FUNCTION WORDS_TO_ARR08B_BE (* this Function combines 4 WORDSs to a 8-BYTE Array; Big-Endian-Format (Network Byte Order) *)
  (* Standard: 61499-1; Description: Copyright (c) 2024 HR Agrartechnik GmbH This program and the accompanying materials are made available under the terms of the Eclipse Public License 2.0 which is available at https://www.eclipse.org/legal/epl-2.0/ SPDX-License-Identifier: EPL-2.0 Big-Endian-Format (Network Byte Order) Siemens S7, Modbus TCP (oft), Ethernet Header *)
  (* Version 1.0, 2024-02-22, Franz Höpfinger, HR Agrartechnik GmbH *)
  PACKAGE logiBUS::utils::conversion::arr::reversing;
  IMPORT eclipse4diac::core::TypeHash;
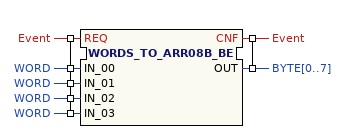
  EVENT_INPUT
    REQ WITH IN_00, IN_01, IN_02, IN_03;
  END_EVENT
  EVENT_OUTPUT
    CNF WITH OUT;
  END_EVENT
  VAR_INPUT
    IN_00 : WORD; (* WORD 00 *)
    IN_01 : WORD; (* WORD 01 *)
    IN_02 : WORD; (* WORD 02 *)
    IN_03 : WORD; (* WORD 03 *)
  END_VAR
  VAR_OUTPUT
    OUT : ARRAY [0..7] OF BYTE; (* ARR08B Output *)
  END_VAR
  BODY IN ST:
PACKAGE logiBUS::utils::conversion::arr::reversing;

(* this Function combines 4 WORDSs to a 8-BYTE Array; Big-Endian-Format (Network Byte Order) *)
FUNCTION WORDS_TO_ARR08B_BE

VAR_INPUT
	IN_00 : WORD; // WORD 00
	IN_01 : WORD; // WORD 01
	IN_02 : WORD; // WORD 02
	IN_03 : WORD; // WORD 03
END_VAR

VAR_OUTPUT
	OUT : ARRAY[0..7] OF BYTE; // ARR08B Output
END_VAR

OUT[0] := IN_00.%B1;
OUT[1] := IN_00.%B0;
OUT[2] := IN_01.%B1;
OUT[3] := IN_01.%B0;
OUT[4] := IN_02.%B1;
OUT[5] := IN_02.%B0;
OUT[6] := IN_03.%B1;
OUT[7] := IN_03.%B0;

END_FUNCTION
  END_BODY
END_FUNCTION
